// TwinCAT 3 PLC project AufgSer3
// ProgramVersion: 3.1.4023.0
// libraries:
//   Tc2_Standard, * (Beckhoff Automation GmbH)
//   Tc2_System, * (Beckhoff Automation GmbH)
//   Tc3_Module, * (Beckhoff Automation GmbH)
// project tree:
//   / PlcTask.TcTTO
//   POUs/ FB_PWM.TcPOU, F_PWM.TcPOU, F_Sine.TcPOU, F_Square.TcPOU, MAIN.TcPOU
// real-time tasks:
//   TASK PlcTask: cycle T#10ms, priority 20, ADS port 350

CONFIGURATION AufgSer3
    RESOURCE PLC ON TwinCAT3
        TASK PlcTask(INTERVAL := T#10ms, PRIORITY := 20);
        PROGRAM MAIN WITH PlcTask : MAIN;
    END_RESOURCE
END_CONFIGURATION

// ---- POUs/MAIN.TcPOU
PROGRAM MAIN
VAR
	// Time
	t				: REAL := 0.0;
	T_task			: INT := 10;  // task cycle time (ms)
	
	// Functions
	ysine			: REAL;
	ysquare			: REAL;
	fbPWM			: FB_PWM;				
	ypwm			: REAL;
END_VAR
VAR CONSTANT
	INT_MAX			: INT := 32767;  // maximum value of integer type
	
END_VAR

// Aufg 1 Sine function
ysine := F_Sine(A := 100.0, yoff := 20.0, w := 2, t := t/1000.0);

// Aufg 2 Square function
ysquare := F_Square(ymax := 100.0, ymin := -100.0, yoff := 20.0, w := 2, t := t/1000.0);

// Aufg 3 PWM function
fbPWM(dutyPct := 25.0, ymax := 100.0, ymin := 0.0, w := 2, t := t/1000.0);
ypwm := fbPWM.y;

// increment time

IF(t+T_task < INT_MAX) THEN
	t := t + T_Task;	
ELSE
	t := 0;
END_IF

END_PROGRAM

// ---- POUs/FB_PWM.TcPOU
FUNCTION_BLOCK FB_PWM
VAR_INPUT
	dutyPct	: REAL;	// Duty cycle (%)
	ymin	: REAL; // Minimalwert
	ymax	: REAL;	// Maximalwert
	w		: REAL; // Kreisfrequenz (rad/s)
	t		: REAL; // Time (s)
END_VAR
VAR_OUTPUT
	y		: REAL; // pwm signal
END_VAR
VAR
	t_elapsed: REAL := 0;  // time since start of pwm cycle [s]
	last_t	: REAL := 0; // time since last call	
	t_cycle	: REAL; // T [s]
	t_duty	: REAL; // time when the duty cycle is over
END_VAR

// add up elapsed time
t_elapsed := t_elapsed + (t - last_t);
last_t := t;

// calc times
t_cycle := (2.0 * 3.14) / w;
t_duty := (dutyPct / 100.0) * t_cycle;

// set new t_start (either when the cylce time is reached or when t_elapsed is negative (failsafe))
IF(t_elapsed > t_cycle OR t_elapsed < 0) THEN
	t_elapsed := 0;
END_IF

// set pwm signal value
IF (t_elapsed > t_duty) THEN
	y := ymin;
ELSE
	y := ymax;
END_IF

END_FUNCTION_BLOCK

// ---- POUs/F_Sine.TcPOU
FUNCTION F_Sine : REAL
VAR_INPUT
	A		: REAL;	// Amplitude
	yoff	: REAL; // offset
	w		: REAL; // Kreisfrequenz (rad/s)
	t		: REAL; // Time (s)
END_VAR
VAR
END_VAR

F_Sine := (A * SIN(w*t)) + yoff;

END_FUNCTION

// ---- POUs/F_Square.TcPOU
FUNCTION F_Square : REAL
VAR_INPUT
	ymin	: REAL;	// Minimalwert
	ymax	: REAL;	// Maximalwert
	yoff	: REAL; // offset
	w		: REAL; // Kreisfrequenz (rad/s)
	t		: REAL; // Time (s)
END_VAR
VAR
	sinRes	: REAL; // sine result
	squareRes: REAL;
END_VAR

sinRes := SIN(w*t);

IF (sinRes > 0) THEN
	squareRes := ymin;
ELSE
	squareRes := ymax;
END_IF

F_Square := squareRes + yoff;

END_FUNCTION

// ---- POUs/F_PWM.TcPOU
FUNCTION F_PWM : REAL
VAR_INPUT
	dutyPct	: REAL;	// Duty cycle (%)
	ymin	: REAL; // Minimalwert
	ymax	: REAL;	// Maximalwert
	w		: REAL; // Kreisfrequenz (rad/s)
	t		: REAL; // Time (s)
END_VAR
VAR
	sinRes	: REAL; // current sin result
	sinResDuty: REAL; // sine result when duty cylce is reached
	t_duty	: REAL; // time when duty cycle is reached
END_VAR

sinRes := SIN(w*t);
t_duty := (dutyPct / 100.0) * ((2.0 * 3.14) / w);
sinResDuty := SIN(w*t_duty);

IF (sinRes > sinResDuty) THEN
	F_PWM := ymin;
ELSE
	F_PWM := ymax;
END_IF

END_FUNCTION
